TYPE ParametersHome :
STRUCT
	Position : LREAL := 10; // in mm
	Mode : MC_HomingMode := MC_DefaultHoming;
END_STRUCT
END_TYPE

(* stored: Version 1.1.0.1, ProductVersion 3.1.4022.10
   POU ParametersHome: Id {1ec44c4d-06f6-4832-b786-9152cf1735f2}, SpecialFunc None *)
